{attribute 'qualified_only'}
VAR_GLOBAL
END_VAR

(* stored: Version 1.1.0.1, ProductVersion 3.1.4022.7
   GVL GVL_07_Alarm_Other: Id {5002bd13-cc3f-4c06-b65c-947c7b27ec10} *)
